# B&R Automation Studio project Zaoshanghaojongwo
Automation Studio 4.5.2.102

## Configuration Config1

### Task classes (Cpu.sw)
```
Cyclic#4:
  Program <- Program.prg
Libraries: Motor
```

### Hardware
```
4PP065_0351_P74 : 4PP065.0351-P74 v1.0.4.0
  Connector IF5:
    ActivateDevice = 1
  ConfigurationID = Zaoshanghaojongwo_Config1
  Simulation = 1
  KeyMappingFile = VC\4PP065_0351_P74.dis
```

## Logical view

### Program Logical/Program (ANSIC)

#### Variables.var
```iecst
VAR
	speed : REAL;
	enable : BOOL;
	counter : INT;
	fb_regulator : FB_Regulator;
	fb_motor1 : FB_Motor;
	fb_motor2 : FB_Motor;
END_VAR
```

#### Cyclic.c
```c
#include <bur/plctypes.h>

#ifdef _DEFAULT_INCLUDES
	#include <AsDefault.h>
#endif

void _CYCLIC ProgramCyclic(void)
{
	if (counter % 200 == 0)
	{
		enable = !enable;
		if (enable)
		{
			speed = 50;
		}
		else
		{
			speed = 0;
		}
	}
	fb_regulator.e = speed - fb_motor1.w;
	FB_Regulator(&fb_regulator);

	fb_motor1.u = fb_regulator.u;
	FB_Motor(&fb_motor1);
	fb_motor2.u = speed * fb_motor2.ke;
	FB_Motor(&fb_motor2);
	counter += 1;
}
```

#### Init.c
```c
#include <bur/plctypes.h>

#ifdef _DEFAULT_INCLUDES
	#include <AsDefault.h>
#endif

void _INIT ProgramInit(void)
{
	fb_regulator.dt = 0.1;
	fb_regulator.integrator.dt = 0.1;
	fb_regulator.max_abs_value = 20.0;
	fb_regulator.k_p = 0.095;
	fb_regulator.k_i = 2.0;
	fb_motor1.dt = 0.1;
	fb_motor1.integrator.dt = 0.1;
	fb_motor1.Tm = 0.063;
	fb_motor1.ke = 0.087;
	fb_motor1.u = 0;
	fb_motor2.dt = 0.1;
	fb_motor2.integrator.dt = 0.1;
	fb_motor2.Tm = 0.063;
	fb_motor2.ke = 0.087;
	fb_motor2.u = 0;
	counter = 0;
	speed = 0;
	enable = 0;
}
```

### Library Logical/Motor (ANSIC)

#### Motor.fun - Exported functions and function blocks
```iecst
{REDUND_ERROR} FUNCTION_BLOCK FB_Motor (*TODO: Add your comment here*) (*$GROUP=User,$CAT=User,$GROUPICON=User.png,$CATICON=User.png*)
	VAR_INPUT
		u : {REDUND_UNREPLICABLE} REAL;
	END_VAR
	VAR_OUTPUT
		w : REAL;
		phi : REAL;
	END_VAR
	VAR
		integrator : FB_Integrator;
		ke : REAL;
		Tm : REAL;
		dt : REAL;
	END_VAR
END_FUNCTION_BLOCK

{REDUND_ERROR} FUNCTION_BLOCK FB_Integrator (*TODO: Add your comment here*) (*$GROUP=User,$CAT=User,$GROUPICON=User.png,$CATICON=User.png*)
	VAR_INPUT
		in : REAL;
	END_VAR
	VAR_OUTPUT
		out : REAL;
	END_VAR
	VAR
		dt : REAL;
	END_VAR
END_FUNCTION_BLOCK

{REDUND_ERROR} FUNCTION_BLOCK FB_Regulator (*TODO: Add your comment here*) (*$GROUP=User,$CAT=User,$GROUPICON=User.png,$CATICON=User.png*)
	VAR_INPUT
		e : {REDUND_UNREPLICABLE} REAL;
	END_VAR
	VAR_OUTPUT
		u : REAL;
	END_VAR
	VAR
		k_p : REAL;
		k_i : REAL;
		integrator : FB_Integrator;
		iyOld : REAL;
		max_abs_value : REAL;
		dt : REAL;
	END_VAR
END_FUNCTION_BLOCK
```

#### FB_Motor.c
```c
#include <bur/plctypes.h>
#ifdef __cplusplus
	extern "C"
	{
#endif
	#include "Motor.h"
#ifdef __cplusplus
	};
#endif
/* TODO: Add your comment here */
void FB_Motor(struct FB_Motor* inst)
{
	inst->integrator.out = inst->w;
	inst->integrator.in = (inst->u/inst->ke - inst->w) * (inst->dt/inst->Tm);
	FB_Integrator(&inst->integrator);
	inst->integrator.in = inst->w = inst->integrator.out;
	inst->integrator.in *= inst->dt;
	inst->integrator.out = inst->phi;
	FB_Integrator(&inst->integrator);
	inst->phi = inst->integrator.out;

}
```

#### FB_Regulator.c
```c
#include <bur/plctypes.h>
#ifdef __cplusplus
	extern "C"
	{
#endif
	#include "Motor.h"
#ifdef __cplusplus
	};
#endif
/* TODO: Add your comment here */
void FB_Regulator(struct FB_Regulator* inst)
{
	REAL a = inst->e * inst->k_p;
	REAL b = inst->e * inst->k_i * inst->dt;
	a = a > inst->max_abs_value ? inst->max_abs_value : a;
	a = a < -inst->max_abs_value ? -inst->max_abs_value : a;
	inst->integrator.in = b + inst->iyOld;
	FB_Integrator(&inst->integrator);
	REAL sum = a + inst->integrator.out;
	inst->u = sum;
	inst->u = inst->u > inst->max_abs_value ? inst->max_abs_value : inst->u;
	inst->u = inst->u < -inst->max_abs_value ? -inst->max_abs_value : inst->u;
	inst->iyOld = inst->u - sum;

}
```

#### FB_Integrator.c
```c
#include <bur/plctypes.h>
#ifdef __cplusplus
	extern "C"
	{
#endif
	#include "Motor.h"
#ifdef __cplusplus
	};
#endif
/* TODO: Add your comment here */
void FB_Integrator(struct FB_Integrator* inst)
{
	inst->out = inst->in * inst->dt + inst->out;
	/*TODO: Add your code here*/
}
```

Listed in the project but not available here: Logical/Global.typ, Logical/Global.var, Logical/Libraries, Logical/Motor/Types.typ, Logical/Motor/Constants.var
